TYPE DUT_TerminalError :
STRUCT
	//Error system related
	iTerminalID : INT;					//ID of the terminal
	Error_ID : ULINT := 0;				//ID for the Error entry
	ErrorState : DUT_ErrorState;		//State of the error
	
	//Error related
	sDateTimeOn : STRING(24);			//Date and time when the error occured. Readable format
	sDateTimeOff : STRING(24);			//Date and time when the error disapeared. Readable format
	sErrorMessage : STRING (128);		//Error message corresponding to WcState and InfoData.State
	ErrorType : INT; 					//Error types (priorities) need to be developed
END_STRUCT
END_TYPE

(* stored: Version 1.1.0.1, ProductVersion 3.1.4022.10
   DUT DUT_TerminalError: Id {8f84cc80-708c-4401-8591-6bfbf208dfab} *)
